TYPE St_days :
STRUCT
	days : ARRAY [1..31] OF REAL;
	fSumDays : REAL;
END_STRUCT
END_TYPE

(* stored: Version 1.1.0.1, ProductVersion 3.1.4024.12
   DUT St_days: Id {99267dd5-0997-4859-a71f-d5100994bd1b} *)
